INTERFACE ICollection EXTENDS IEnumerable

{attribute 'OPC.UA.DA.Property' := '1'}
{attribute 'monitoring' := 'call'}
PROPERTY Count : DINT
GET
END_GET
END_PROPERTY

END_INTERFACE

(* stored: Version 1.1.0.1
   Itf ICollection: Id {ded0232e-5c0d-07b7-1848-d72cdabf5069}
   Property Count: Id {0e912d25-e3c7-0123-2db5-9605b7a8ef9b}
   Get Get: Id {adcfa157-f0c0-0728-3033-0204eb60f2d3} *)
